FUNCTION F_Concat6 : T_MaxString
VAR_INPUT
	sOne : STRING;
	sTwo : STRING;
	sThree : STRING;
	sFour : STRING;
	sFive : STRING;
	sSix : STRING;
END_VAR

F_Concat6 := CONCAT(
					sOne,
					F_Concat5( sTwo, sThree, sFour, sFive, sSix )
				);

END_FUNCTION

(* stored: Version 1.1.0.1, ProductVersion 3.1.4022.9
   POU F_Concat6: Id {f9bdfea7-84cb-4914-a06b-6fcfc4a0418c}, SpecialFunc None *)
